(*udt (user defined type) for Schneider Electric VFD I/O Module
	Author(S): Justin Vandongen of Sodecia GTAC;

------------------------------------------------------------------------
	REVISION NOTES:

	Version 20180808
		- Initial Concept, j.vandongen
		- tested on ATV320 v1.11 ethercat module from schneider, j.vandongen
	Version 20190123
		- re-organized for more consistancy to generic device udts, b.lekx-toniolo

------------------------------------------------------------------------
*)

TYPE udt_Schneider_VFD_Inputs_20190123 :
	STRUCT
	InfoData: udt_ECATSlave_StatusEXT;

	Status_Word: UINT;
	Control_Effort: INT;
	Move_Time: TIME;

	END_STRUCT
END_TYPE

(* stored: Version 1.1.0.1, ProductVersion 3.1.4024.5
   DUT udt_Schneider_VFD_Inputs_20190123: Id {7fa81eba-8a39-495e-9b87-e9b3a2354dd8} *)
